FUNCTION_BLOCK FB_SA
VAR_INPUT
END_VAR
VAR_OUTPUT
END_VAR
VAR
END_VAR

END_FUNCTION_BLOCK

(* stored: Version 1.1.0.1
   POU FB_SA: Id {d63b48a3-aa8f-4dc5-8329-9b7378936e32}, SpecialFunc None *)
